INTERFACE ITF_BA_AMR

METHOD MC_ChangeSpeedOverride : INT
VAR_INPUT
	factor: REAL;
END_VAR
END_METHOD

METHOD MC_MoveAxesAbsolute : BOOL
VAR_INPUT
	target: stTarget3D;
END_VAR
END_METHOD

METHOD MC_MoveAxesRelative : BOOL
VAR_INPUT
	axes: ARRAY[1..6] OF FB_Axis;
	offsets: ARRAY[1..6] OF REAL;
END_VAR
END_METHOD

METHOD MC_MoveLinearAbsolute : BOOL
VAR_INPUT
	target: stTarget3D;
END_VAR
END_METHOD

METHOD PUBLIC MC_ReadAnalogInput : LREAL
VAR_INPUT
	input : INT;
END_VAR
END_METHOD

METHOD PUBLIC MC_ReadDigitalInput : BOOL
VAR_INPUT
	input : INT;
END_VAR
END_METHOD

METHOD PUBLIC MC_SetDigitalOutput : BOOL
VAR_INPUT
	output : INT;
	value : BOOL;
END_VAR
END_METHOD

METHOD PUBLIC MC_SetOperationMode : BOOL
VAR_INPUT
	mode: eMode;
END_VAR
END_METHOD

END_INTERFACE

(* stored: Version 1.1.0.1, ProductVersion 3.1.4026.18
   Itf ITF_BA_AMR: Id {4d7b847a-995a-4492-b7ff-3c61a44f7325}
   Method MC_ChangeSpeedOverride: Id {bd1956a8-a155-4695-8b02-2ec96a217abb}
   Method MC_MoveAxesAbsolute: Id {ab8630f6-1bed-432f-ad06-bc8c41fbe76e}
   Method MC_MoveAxesRelative: Id {902d67bf-6067-419a-b02e-8f921433ee19}
   Method MC_MoveLinearAbsolute: Id {e0a6e723-237e-46f4-b289-eb3bd8fdd16f}
   Method MC_ReadAnalogInput: Id {070b53ff-9723-48be-8892-9dc9abcc79fb}
   Method MC_ReadDigitalInput: Id {ccb9b97c-0b1b-4da0-ac89-c4217398f24e}
   Method MC_SetDigitalOutput: Id {a42b56c3-97da-4208-abed-8bbbaf37cf4f}
   Method MC_SetOperationMode: Id {49aaee93-8cbe-40c8-a610-36f8e4973d32} *)
